KUKA KRL data list: MillingProgram1.dat

&ACCESS RV
DEFDAT MillingProgram1 PUBLIC

ENDDAT
